Omron Sysmac Studio project Compare (Sysmac Studio 1.65.0.64007, StandardProject)

# Controller new_Controller_0: NX1P2-1040DT1 version 1.69
Task PrimaryTask (priority 4, period or condition 2000): Program0

VAR_GLOBAL
    TON_ET : TIME;
    Cmp_OUT : BOOL;
END_VAR

PROGRAM Program0
VAR
    deneme : BOOL;
    Real_V : REAL;
    INT_V : INT;
    TON : TON;
END_VAR
VAR_EXTERNAL
    TON_ET : TIME;
    Cmp_OUT : BOOL;
END_VAR

(* Section Section0: ladder, written here as Structured Text *)

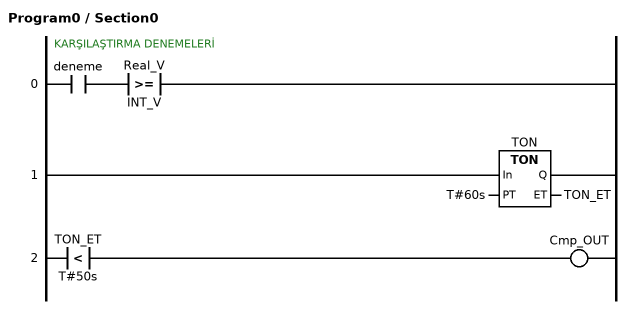
(* Rung 0: KARŞILAŞTIRMA DENEMELERİ *)
(* drawn but driving nothing: deneme, Real_V, INT_V *)
(* Rung 1 *)
TON(In := TRUE, PT := T#60s, ET => TON_ET);
(* Rung 2 *)
Cmp_OUT := TON_ET < T#50s;
END_PROGRAM